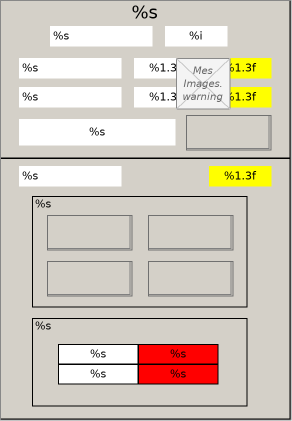
VISUALIZATION VISU_IC6  // 292x421
VAR_IN_OUT
	M_Input_Ctrl:		BLOCK_IC6;
	M_Input_QZ1:		BLOCK_XTAL;
	M_Input_QZ2:		BLOCK_XTAL;
END_VAR
    GroupBox (0,144 290x275), invisible if: NOT M_Input_Ctrl.VISU_Show_Details
        Rectangle (0,14 290x261)
        RoundedRectangle (32,52 215x111), "%s", text list: 'TextList_IC6', text index: 4
        Button (47,71 85x35), input disabled if: NOT PRG_USER.ACTU_USER.MAINTENANCE OR NOT MACHINE.STATE_Manu, text list: 'TextList_IC6', text index: 5
            toggle M_Input_Ctrl.M_Start
        Button (47,117 85x35), text list: 'TextList_IC6', text index: 6
            toggle M_Input_Ctrl.M_Stop
        Button (148,71 85x35), text list: 'TextList_IC6', text index: 7
            toggle M_Input_Ctrl.M_RAZ_Thick
        Button (148,117 85x35), text list: 'TextList_IC6', text index: 8
            toggle M_Input_Ctrl.M_Reset
        Textfield (19,22 102x20), "%s", text list: 'TextList_IC6', text index: 3
        Textfield (209,22 62x20), "%1.3f", text variable: M_Input_Ctrl.STATE_Puissance
        RoundedRectangle (32,174 215x88), "%s", text list: 'TextList_IC6', text index: 9
        Rectangle (58,200 80x20), "%s", text variable: M_Input_QZ1.MNEMO
        Rectangle (58,220 80x20), "%s", text variable: M_Input_QZ2.MNEMO
        Rectangle (138,200 80x20), "OK", invisible if: M_Input_QZ1.STATE_NOK
        Rectangle (138,200 80x20), "%s", invisible if: NOT M_Input_QZ1.STATE_NOK, text list: 'TextList_IC6', text index: 10
        Rectangle (138,220 80x20), "OK", invisible if: M_Input_QZ2.STATE_NOK
        Rectangle (138,220 80x20), "%s", invisible if: NOT M_Input_QZ2.STATE_NOK, text list: 'TextList_IC6', text index: 10
    Rectangle (0,0 290x158), "%s", text variable: M_Input_Ctrl.MNEMO
    Textfield (19,58 102x20), "%s", text list: 'TextList_IC6', text index: 0
    Textfield (19,87 102x20), "%s", text list: 'TextList_IC6', text index: 1
    Textfield (209,58 62x20), "%1.3f", text variable: M_Input_Ctrl.STATE_Global_Rate
    Textfield (209,87 62x20), "%1.3f", text variable: M_Input_Ctrl.STATE_Global_Thick
    Textfield (134,58 62x20), "%1.3f", text variable: M_Input_Ctrl.I_Rate_App
    Textfield (134,87 62x20), "%1.3f", text variable: M_Input_Ctrl.I_Epaisseur
    RoundedRectangle (19,119 156x26), "%s", text variable: M_Input_Ctrl.STATE_Phase
    Image (176,58 54x51), invisible if: NOT M_Input_Ctrl.STATE_NOK, image: MesImages.warning
    Button (186,115 85x35), text list: 'TextList_IC6', text index: 2
        toggle M_Input_Ctrl.VISU_Show_Details
    Textfield (50,26 102x20), "%s", text list: 'TextList_IC6', text index: 11
    Textfield (165,26 62x20), "%i", text variable: M_Input_Ctrl.PRM_Materiau, input disabled if: MACHINE.STATE_Prod
        OnMouseClick: write the text variable via Default, min 1, max 6
END_VISUALIZATION

(* stored: Version 1.1.0.1, ProductVersion 3.1.4024.10
   Visu VISU_IC6: Id {2e81b219-8b79-4395-8cf6-ec7c076f15a8} *)
